// TIA Portal V20 export
VAR_GLOBAL   // PLC tag table "Unit1"
   "BA010AZCRMP101.00" AT %I100.0 : Bool;   // MOTOR POWER TRIPPED E202CB
   "BA010AZCRMP101.01" AT %I100.1 : Bool;   // REELCUT CONVEYOR RING BLOW POWER TRIPPED
   "BA010AZCRMP101.02" AT %I100.2 : Bool;   // STACKING-1 CONVEYOR RING BLOW POWER TRIPPED E214CB
   "BA010AZCRMP101.03" AT %I100.3 : Bool;   // STACKING-2 CONVEYOR RING BLOW POWER TRIPPED E220CB
   "BA010AZCRMP101.04" AT %I100.4 : Bool;   // SPARE
   "BA010AZCRMP101.05" AT %I100.5 : Bool;   // E6404PWS CONTROLLER POWER SMPS AC POWER TRIPPED E320CB
   "BA010AZCRMP101.06" AT %I100.6 : Bool;   // E6704PWS CONTROLLER POWER SMPS AC POWER TRIPPED E326CB
   "BA010AZCRMP101.07" AT %I100.7 : Bool;   // E6804PWS SAFETY POWER SMPS AC POWER TRIPPED E332CB
   "BA010AZCRMP101.10" AT %I101.0 : Bool;   // SPARE
   "BA010AZCRMP101.11" AT %I101.1 : Bool;   // POWER METER POWER TRIPPED E720CB
   "BA010AZCRMP101.12" AT %I101.2 : Bool;   // POWER METER CONTROL POWER TRIPPED E726CB
   "BA010AZCRMP101.13" AT %I101.3 : Bool;   // SPARE
   "BA010AZCRMP101.14" AT %I101.4 : Bool;   // PROCESSOR POWER ON TRIPPED E4116CB
   "BA010AZCRMP101.15" AT %I101.5 : Bool;   // PROGRAMMING POWER OUTLET TRIPPED E4156CB
   "BA010AZCRMP101.16" AT %I101.6 : Bool;   // SPARE
   "BA010AZCRMP101.17" AT %I101.7 : Bool;   // PANEL LED POWER TRIPPED E4304CB
   "BA010AZCRMP101.20" AT %I102.0 : Bool;   // SPARE
   "BA010AZCRMP101.21" AT %I102.1 : Bool;   // PLC POWER SMPS DC OK E4404PWS
   "BA010AZCRMP101.22" AT %I102.2 : Bool;   // CONTROL LEVEL HUB POWER TRIPPED E4420CB
   "BA010AZCRMP101.23" AT %I102.3 : Bool;   // MAIN HMI POWER TRIPPED E4426CB
   "BA010AZCRMP101.24" AT %I102.4 : Bool;   // PORTABLE HMI POWER TRIPPED E4432CB
   "BA010AZCRMP101.25" AT %I102.5 : Bool;   // PORTABLE HMI POWER TRIPPED E4456CB
   "BA010AZCRMP101.26" AT %I102.6 : Bool;   // SPARE
   "BA010AZCRMP101.27" AT %I102.7 : Bool;   // SPARE
   "BA010AZCRMP101.30" AT %I103.0 : Bool;   // 120VAC CONTROL POWER TR PRIMARY TRIPPED E5100CB
   "BA010AZCRMP101.31" AT %I103.1 : Bool;   // 120VAC CONTROL POWER TR SECONDARY TRIPPED E5110CB
   "BA010AZCRMP101.32" AT %I103.2 : Bool;   // CONTROL POWER ON TRIPPED E5116CB
   "BA010AZCRMP101.33" AT %I103.3 : Bool;   // VISION MONITOR POWER STRIP OUTLET POWER TRIPPED E5160CB
   "BA010AZCRMP101.34" AT %I103.4 : Bool;   // MCU & RFD HANDY POWER STRIP OUTLET POWER TRIPPED E5166CB
   "BA010AZCRMP101.35" AT %I103.5 : Bool;   // VISION LIGHT CONTROLLER POWER STRIP OUTLET POWER TRIPPED E5172CB
   "BA010AZCRMP101.36" AT %I103.6 : Bool;   // SPARE
   "BA010AZCRMP101.37" AT %I103.7 : Bool;   // FFU POWER-1 POWER TRIPPED E3222CB
   "BA010AZCRMP102.00" AT %I104.0 : Bool;   // SPARE
   "BA010AZCRMP102.01" AT %I104.1 : Bool;   // CONTROL POWER SMPS DC OK E6104PWS
   "BA010AZCRMP102.02" AT %I104.2 : Bool;   // ET200MP I/O OUTPUT POWER TRIPPED E6154CB
   "BA010AZCRMP102.03" AT %I104.3 : Bool;   // JUNCTION BOX CONTROL POWER TRIPPED E6180CB
   "BA010AZCRMP102.04" AT %I104.4 : Bool;   // CLASS 2 SMPS POWER TRIPPED E6204CB
   "BA010AZCRMP102.05" AT %I104.5 : Bool;   // CLASS 2 SMPS MONITORING E6206PWS
   "BA010AZCRMP102.06" AT %I104.6 : Bool;   // ET200ECO PN-1 POWER TRIPPED E6220CB
   "BA010AZCRMP102.07" AT %I104.7 : Bool;   // ET200ECO PN-2 POWER TRIPPED E6224CB
   "BA010AZCRMP102.10" AT %I105.0 : Bool;   // ET200ECO PN-3 POWER TRIPPED E6228CB
   "BA010AZCRMP102.11" AT %I105.1 : Bool;   // SPARE
   "BA010AZCRMP102.12" AT %I105.2 : Bool;   // PANEL FAN POWER TRIPPED E6304CB
   "BA010AZCRMP102.13" AT %I105.3 : Bool;   // SPARE
   "BA010AZCRMP102.14" AT %I105.4 : Bool;   // CONTROLLER POWER SMPS DC OK E6404PWS
   "BA010AZCRMP102.15" AT %I105.5 : Bool;   // CONTROLLER DC POWER TRIPPED E6406CB
   "BA010AZCRMP102.16" AT %I105.6 : Bool;   // SERVO CONTROL POWER TRIPPED E6416CB
   "BA010AZCRMP102.17" AT %I105.7 : Bool;   // MANIFOLD-1 CONTROL POWER TRIPPED E6422CB
   "BA010AZCRMP102.20" AT %I106.0 : Bool;   // SPARE
   "BA010AZCRMP102.21" AT %I106.1 : Bool;   // RFID POWER TRIPPED E6456CB
   "BA010AZCRMP102.22" AT %I106.2 : Bool;   // QR READER POWER TRIPPED E6462CB
   "BA010AZCRMP102.23" AT %I106.3 : Bool;   // QR READER POWER TRIPPED E6468CB
   "BA010AZCRMP102.24" AT %I106.4 : Bool;   // SPARE
   "BA010AZCRMP102.25" AT %I106.5 : Bool;   // SPARE
   "BA010AZCRMP102.26" AT %I106.6 : Bool;   // CONTROLLER POWER SMPS DC OK E6704PWS
   "BA010AZCRMP102.27" AT %I106.7 : Bool;   // CONTROLLER DC POWER TRIPPED E6706CB
   "BA010AZCRMP102.30" AT %I107.0 : Bool;   // HANDY QR READER POWER TRIPPED E6716CB
   "BA010AZCRMP102.31" AT %I107.1 : Bool;   // VISION CONTROLLER POWER TRIPPED E6722CB
   "BA010AZCRMP102.32" AT %I107.2 : Bool;   // LINE LASER MODULE-1 POWER TRIPPED E6728CB
   "BA010AZCRMP102.33" AT %I107.3 : Bool;   // LINE LASER MODULE-2 POWER TRIPPED E6734CB
   "BA010AZCRMP102.34" AT %I107.4 : Bool;   // EPC CONTROLLER-1 POWER TRIPPED E6756CB
   "BA010AZCRMP102.35" AT %I107.5 : Bool;   // EPC CONTROLLER-2 POWER TRIPPED E6762CB
   "BA010AZCRMP102.36" AT %I107.6 : Bool;   // EPC CONTROLLER-3 POWER TRIPPED E6768CB
   "BA010AZCRMP102.37" AT %I107.7 : Bool;   // DRIVE-CLIQ HUB POWER TRIPPED E6774CB
   "BA010AZCRMP103.00" AT %I108.0 : Bool;   // EQUIPMENT LED POWER TRIPPED E6780CB
   "BA010AZCRMP103.01" AT %I108.1 : Bool;   // MOTOR POWER MC COIL POWER TRIPPED E6786CB
   "BA010AZCRMP103.02" AT %I108.2 : Bool;   // SAFETY POWER SMPS DC OK E6804PWS
   "BA010AZCRMP103.03" AT %I108.3 : Bool;   // SAFETY DC POWER TRIPPED E6808CB
   "BA010AZCRMP103.04" AT %I108.4 : Bool;   // ET200SP I/O SAFETY POWER TRIPPED E6816CB
   "BA010AZCRMP103.05" AT %I108.5 : Bool;   // JUNCTION BOX CONTROL POWER TRIPPED E6836CB
   "BA010AZCRMP103.06" AT %I108.6 : Bool;   // ET200ECO PN-SAFETY-1 POWER TRIPPED E6856CB
   "BA010AZCRMP103.07" AT %I108.7 : Bool;   // SPARE
   "BA010AZCRMP103.10" AT %I109.0 : Bool;   // SPARE
   "BA010AZCRMP103.11" AT %I109.1 : Bool;   // SPARE
   "BA010AZCRMP103.12" AT %I109.2 : Bool;   // SPARE
   "BA010AZCRMP103.13" AT %I109.3 : Bool;   // SPARE
   "BA010AZCRMP103.14" AT %I109.4 : Bool;   // SPARE
   "BA010AZCRMP103.15" AT %I109.5 : Bool;   // SPARE
   "BA010AZCRMP103.16" AT %I109.6 : Bool;   // SPARE
   "BA010AZCRMP103.17" AT %I109.7 : Bool;   // SPARE
   "BA010AZCRMP103.20" AT %I110.0 : Bool;   // SPARE
   "BA010AZCRMP103.21" AT %I110.1 : Bool;   // SPARE
   "BA010AZCRMP103.22" AT %I110.2 : Bool;   // SPARE
   "BA010AZCRMP103.23" AT %I110.3 : Bool;   // SPARE
   "BA010AZCRMP103.24" AT %I110.4 : Bool;   // SPARE
   "BA010AZCRMP103.25" AT %I110.5 : Bool;   // SPARE
   "BA010AZCRMP103.26" AT %I110.6 : Bool;   // SPARE
   "BA010AZCRMP103.27" AT %I110.7 : Bool;   // SPARE
   "BA010AZCRMP103.30" AT %I111.0 : Bool;   // SPARE
   "BA010AZCRMP103.31" AT %I111.1 : Bool;   // SPARE
   "BA010AZCRMP103.32" AT %I111.2 : Bool;   // SPARE
   "BA010AZCRMP103.33" AT %I111.3 : Bool;   // SPARE
   "BA010AZCRMP103.34" AT %I111.4 : Bool;   // SPARE
   "BA010AZCRMP103.35" AT %I111.5 : Bool;   // SPARE
   "BA010AZCRMP103.36" AT %I111.6 : Bool;   // SPARE
   "BA010AZCRMP103.37" AT %I111.7 : Bool;   // SPARE
   "BA010AZCRSP201.00" AT %I700.0 : Bool;   // AUTO INITIATE PBL (GREEN)
   "BA010AZCRSP201.01" AT %I700.1 : Bool;   // STOP PBL (RED)
   "BA010AZCRSP201.02" AT %I700.2 : Bool;   // SPARE
   "BA010AZCRSP201.03" AT %I700.3 : Bool;   // SPARE
   "BA010AZCRSP201.04" AT %I700.4 : Bool;   // SPARE
   "BA010AZCRSP201.05" AT %I700.5 : Bool;   // SPARE
   "BA010AZCRSP201.06" AT %I700.6 : Bool;   // SPARE
   "BA010AZCRSP201.07" AT %I700.7 : Bool;   // SPARE
   "BA010AZCRSP201.10" AT %I701.0 : Bool;   // MAIN HMI POWER TRIPPED E110CB
   "BA010AZCRSP201.11" AT %I701.1 : Bool;   // SPARE
   "BA010AZCRSP201.12" AT %I701.2 : Bool;   // SPARE
   "BA010AZCRSP201.13" AT %I701.3 : Bool;   // SPARE
   "BA010AZCRSP201.14" AT %I701.4 : Bool;   // SPARE
   "BA010AZCRSP201.15" AT %I701.5 : Bool;   // SPARE
   "BA010AZCRSP201.16" AT %I701.6 : Bool;   // SPARE
   "BA010AZCRSP201.17" AT %I701.7 : Bool;   // SPARE
   BA010AZCRCU1_Actor_Interface_AddressIn AT %I5000.0 : "LPD_typePDTel390In";
   BA010AZCRCU2_Actor_Interface_AddressIn AT %I5004.0 : "LPD_typePDTel390In";
   BA010AZCRCU3_Actor_Interface_AddressIn AT %I5011.0 : "LPD_typePDTel390In";
   BA010AZCRSLM_Actor_Interface_AddressIn AT %I5050.0 : "LPD_typePDTel370In";
   "BA010AZCRMP104.00" AT %Q100.0 : Bool;   // EQUIPMENT LED LAMP RELAY ON
   "BA010AZCRMP104.01" AT %Q100.1 : Bool;   // SPARE
   "BA010AZCRMP104.02" AT %Q100.2 : Bool;   // SPARE
   "BA010AZCRMP104.03" AT %Q100.3 : Bool;   // CLASS2 SMPS ALARM RESET
   "BA010AZCRMP104.04" AT %Q100.4 : Bool;   // SPARE
   "BA010AZCRMP104.05" AT %Q100.5 : Bool;   // SPARE
   "BA010AZCRMP104.06" AT %Q100.6 : Bool;   // SPARE
   "BA010AZCRMP104.07" AT %Q100.7 : Bool;   // SPARE
   "BA010AZCRMP104.10" AT %Q101.0 : Bool;   // SPARE
   "BA010AZCRMP104.11" AT %Q101.1 : Bool;   // SPARE
   "BA010AZCRMP104.12" AT %Q101.2 : Bool;   // SPARE
   "BA010AZCRMP104.13" AT %Q101.3 : Bool;   // SPARE
   "BA010AZCRMP104.14" AT %Q101.4 : Bool;   // SPARE
   "BA010AZCRMP104.15" AT %Q101.5 : Bool;   // SPARE
   "BA010AZCRMP104.16" AT %Q101.6 : Bool;   // SPARE
   "BA010AZCRMP104.17" AT %Q101.7 : Bool;   // SPARE
   "BA010AZCRMP104.20" AT %Q102.0 : Bool;   // SPARE
   "BA010AZCRMP104.21" AT %Q102.1 : Bool;   // SPARE
   "BA010AZCRMP104.22" AT %Q102.2 : Bool;   // SPARE
   "BA010AZCRMP104.23" AT %Q102.3 : Bool;   // SPARE
   "BA010AZCRMP104.24" AT %Q102.4 : Bool;   // SPARE
   "BA010AZCRMP104.25" AT %Q102.5 : Bool;   // SPARE
   "BA010AZCRMP104.26" AT %Q102.6 : Bool;   // SPARE
   "BA010AZCRMP104.27" AT %Q102.7 : Bool;   // SPARE
   "BA010AZCRMP104.30" AT %Q103.0 : Bool;   // SPARE
   "BA010AZCRMP104.31" AT %Q103.1 : Bool;   // SPARE
   "BA010AZCRMP104.32" AT %Q103.2 : Bool;   // SPARE
   "BA010AZCRMP104.33" AT %Q103.3 : Bool;   // SPARE
   "BA010AZCRMP104.34" AT %Q103.4 : Bool;   // SPARE
   "BA010AZCRMP104.35" AT %Q103.5 : Bool;   // SPARE
   "BA010AZCRMP104.36" AT %Q103.6 : Bool;   // SPARE
   "BA010AZCRMP104.37" AT %Q103.7 : Bool;   // SPARE
   "BA010AZCRSP202.00" AT %Q700.0 : Bool;   // AUTO INITIATE PBL LAMP ON (GREEN)
   "BA010AZCRSP202.01" AT %Q700.1 : Bool;   // STOP PBL LAMP ON (RED)
   "BA010AZCRSP202.02" AT %Q700.2 : Bool;   // RESERVE
   "BA010AZCRSP202.03" AT %Q700.3 : Bool;   // ENABLE PBL LAMP ON (BLACK)
   "BA010AZCRSP202.04" AT %Q700.4 : Bool;   // SAFETY RESET PBL LAMP ON (BLUE)
   "BA010AZCRSP202.05" AT %Q700.5 : Bool;   // SPARE
   "BA010AZCRSP202.06" AT %Q700.6 : Bool;   // SPARE
   "BA010AZCRSP202.07" AT %Q700.7 : Bool;   // SPARE
   "BA010AZCRSP202.10" AT %Q701.0 : Bool;   // TOWER LAMP 1 ON (RED)
   "BA010AZCRSP202.11" AT %Q701.1 : Bool;   // TOWER LAMP 2 ON (AMBER)
   "BA010AZCRSP202.12" AT %Q701.2 : Bool;   // TOWER LAMP 3 ON (GREEN)
   "BA010AZCRSP202.13" AT %Q701.3 : Bool;   // TOWER LAMP 4 ON (WHITE)
   "BA010AZCRSP202.14" AT %Q701.4 : Bool;   // TOWER LAMP 5 ON (BLUE)
   "BA010AZCRSP202.15" AT %Q701.5 : Bool;   // TOWER LAMP 6 ON (BUZZER)
   "BA010AZCRSP202.16" AT %Q701.6 : Bool;   // SPARE
   "BA010AZCRSP202.17" AT %Q701.7 : Bool;   // SPARE
   BA010AZCRCU1_Actor_Interface_AddressOut AT %Q5000.0 : "LPD_typePDTel390Out";
   BA010AZCRCU2_Actor_Interface_AddressOut AT %Q5004.0 : "LPD_typePDTel390Out";
   BA010AZCRCU3_Actor_Interface_AddressOut AT %Q5011.0 : "LPD_typePDTel390Out";
   BA010AZCRSLM_Actor_Interface_AddressOut AT %Q5050.0 : "LPD_typePDTel370Out";
   "BA010AZCRSP501.00" AT %I3000.0 : Bool;   // CONTROL DC POWER TRIPPED E156CB
   "BA010AZCRSP501.01" AT %I3000.1 : Bool;   // SAFETY DC POWER TRIPPED E218CB
   "BA010AZCRBK03.03" AT %I1008.3 : Bool;   // DIGITAL PRESSURE SWITCH OUT1
   "BA010AZCRBK03.13" AT %I1009.3 : Bool;   // DIGITAL PRESSURE SWITCH OUT2
END_VAR
VAR_GLOBAL CONSTANT   // user constants
   U1_NO_OF_EMs : Int := 7;   // Highest Value of equipment modules in the unit (Counting starts from 0)
   U1_EM0 : Int := 0;   // Equipment Module 0
   U1_EM1 : Int := 1;   // Equipment Module 1
   U1_EM2 : Int := 2;   // Equipment Module 2
   U1_EM3 : Int := 3;   // Equipment Module 3
   U1_EM4 : Int := 4;   // Equipment Module 4
   U1_EM5 : Int := 5;   // Equipment Module 5
   U1_EM6 : Int := 6;   // Equipment Module 6
   U1_EM7 : Int := 7;   // Equipment Module 7
END_VAR
